TYPE ST_vaederdata :
STRUCT
	name: STRING;
	levelType: STRING;
	level: REAL;
	unit: STRING;
	values: ARRAY[0..0] OF REAL;
	
END_STRUCT
END_TYPE

(* stored: Version 1.1.0.1, ProductVersion 3.1.4024.12
   DUT ST_vaederdata: Id {1b787647-6478-4e28-9387-5c2c55663c7d} *)
